Omron CX-Programmer project 新工程 (CX-Programmer 9.42)

# PLC 新PLC1: CP1H XA

## Global symbols (name address type ; comment)
0.00 BOOL  ; 开始
0.01 BOOL  ; 复位
10.01 BOOL  ; s1
10.02 BOOL  ; s2
10.03 BOOL  ; s3
10.04 BOOL  ; s4

## Program 新程序1 (cyclic task 0)

### Section 段1

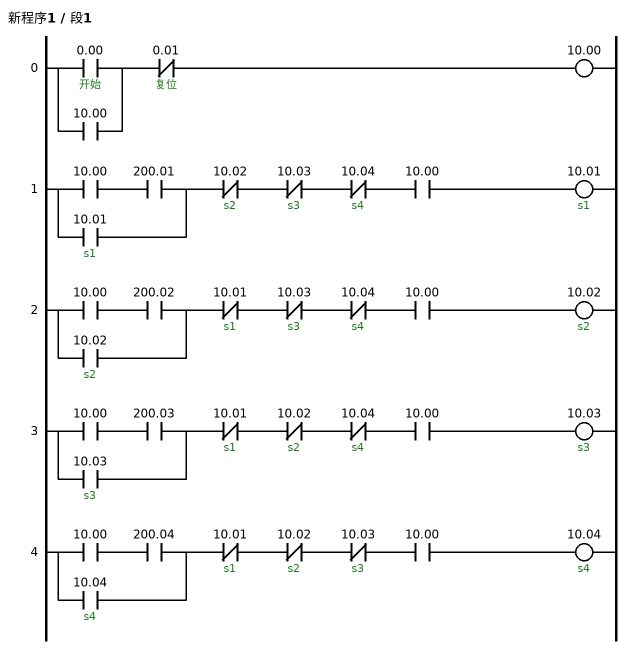
; rung 0
LD 0.00  ; 开始
OR 10.00
ANDNOT 0.01  ; 复位
OUT 10.00
; rung 1
LD 10.00
AND 200.01
OR 10.01  ; s1
ANDNOT 10.02  ; s2
ANDNOT 10.03  ; s3
ANDNOT 10.04  ; s4
AND 10.00
OUT 10.01  ; s1
; rung 2
LD 10.00
AND 200.02
OR 10.02  ; s2
ANDNOT 10.01  ; s1
ANDNOT 10.03  ; s3
ANDNOT 10.04  ; s4
AND 10.00
OUT 10.02  ; s2
; rung 3
LD 10.00
AND 200.03
OR 10.03  ; s3
ANDNOT 10.01  ; s1
ANDNOT 10.02  ; s2
ANDNOT 10.04  ; s4
AND 10.00
OUT 10.03  ; s3
; rung 4
LD 10.00
AND 200.04
OR 10.04  ; s4
ANDNOT 10.01  ; s1
ANDNOT 10.02  ; s2
ANDNOT 10.03  ; s3
AND 10.00
OUT 10.04  ; s4

### Section END
; rung 0
END(001)